TYPE stStationStatus :
STRUCT
	Empty : BOOL;
	Complete : BOOL;
	Operating : BOOL;
	Ready : BOOL;
	HasMover : BOOL;
END_STRUCT
END_TYPE

(* stored: Version 1.1.0.1
   DUT stStationStatus: Id {ceb7c38e-5cf7-43c2-b991-d63b777bc2dc} *)
